Staubli VAL3: findNumberInMatrix.pgx

program findNumberInMatrix(num& x_nInput[] (dimensions=2), num x_nNumber, num& x_nIndexX[], num& x_nIndexY[], bool& x_bFound)
  local num l_nX
  local num l_nY
  local num l_nFoundCounter
begin

  resize(x_nIndexX,1,1)
  x_nIndexX = -1
  resize(x_nIndexY,1,1)
  x_nIndexY = -1
  x_bFound = false

  for l_nX = 0 to size(x_nInput,1)-1
    for l_nY = 0 to size(x_nInput,2)-1

      if x_nNumber == x_nInput[l_nX,l_nY]
        x_bFound = true
        if l_nFoundCounter != 0
          append(x_nIndexX)
          append(x_nIndexY)
        endIf

        x_nIndexX[l_nFoundCounter] = l_nX
        x_nIndexY[l_nFoundCounter] = l_nY
        l_nFoundCounter = l_nFoundCounter + 1
      endIf

    endFor
  endFor


end
